// TIA Portal V18 export
FUNCTION_BLOCK "SearchArea_2doors"   // FB8, LAD
{ S7_Optimized_Access := 'TRUE' }
VERSION : 0.1
// stored: AutoNumber true, IsIECCheckEnabled false, IsRetainMemResEnabled false, MemoryReserve 100, SetENOAutomatically false, UDAEnableTagReadback false
   VAR_INPUT
      SB1 : Bool;
      SB2 : Bool;
      Door1 : Bool;
      Door2 : Bool;
      "E-Stop" : Bool;
      SearchArea_Time : Time := T#5m;
      Reset : Bool;
   END_VAR
   VAR
      SearchArea_Timer { S7_SetPoint := 'True'} : TON_TIME;
      SearchArea_Status : Int;   // 0:未搜索;1:搜索中;2:搜索完成;
      "Step" { S7_SetPoint := 'True'} : Int;
      Error { ExternalAccessible := 'False'; ExternalVisible := 'False'; ExternalWritable := 'False'} : Struct
         All { ExternalAccessible := 'False'; ExternalVisible := 'False'; ExternalWritable := 'False'} : Bool;   // 搜索总故障
         StartFail { ExternalAccessible := 'False'; ExternalVisible := 'False'; ExternalWritable := 'False'} : Bool;   // 搜索启动失败，请确认未按下搜索按钮2或未关闭门1或门2
         WrongSequence1 { ExternalAccessible := 'False'; ExternalVisible := 'False'; ExternalWritable := 'False'} : Bool;   // 搜索顺序错误，此时应按下搜索按钮2，请勿按搜索按钮1或关闭门1或门2
         WrongSequence2 { ExternalAccessible := 'False'; ExternalVisible := 'False'; ExternalWritable := 'False'} : Bool;   // 搜索顺序错误，此时应关闭门1，请勿按搜索按钮1或搜索按钮2或门2
         WrongSequence3 { ExternalAccessible := 'False'; ExternalVisible := 'False'; ExternalWritable := 'False'} : Bool;   // 搜索顺序错误，此时应关闭门2，请勿按搜索按钮1或搜索按钮2或打开门1
         Timeout { ExternalAccessible := 'False'; ExternalVisible := 'False'; ExternalWritable := 'False'} : Bool;   // 搜索超时
      END_STRUCT;
   END_VAR
   VAR_TEMP   // added for the SCL form of the ladder/FBD networks
      _w1 : Bool;
   END_VAR
BEGIN

REGION Network 1: 搜索破坏
   // 搜索完成后，当搜索按钮按下，门被打开，急停按钮按下，搜索状态设置为未搜索
   // 需与客户确认破坏条件是否包含搜索按钮和急停？
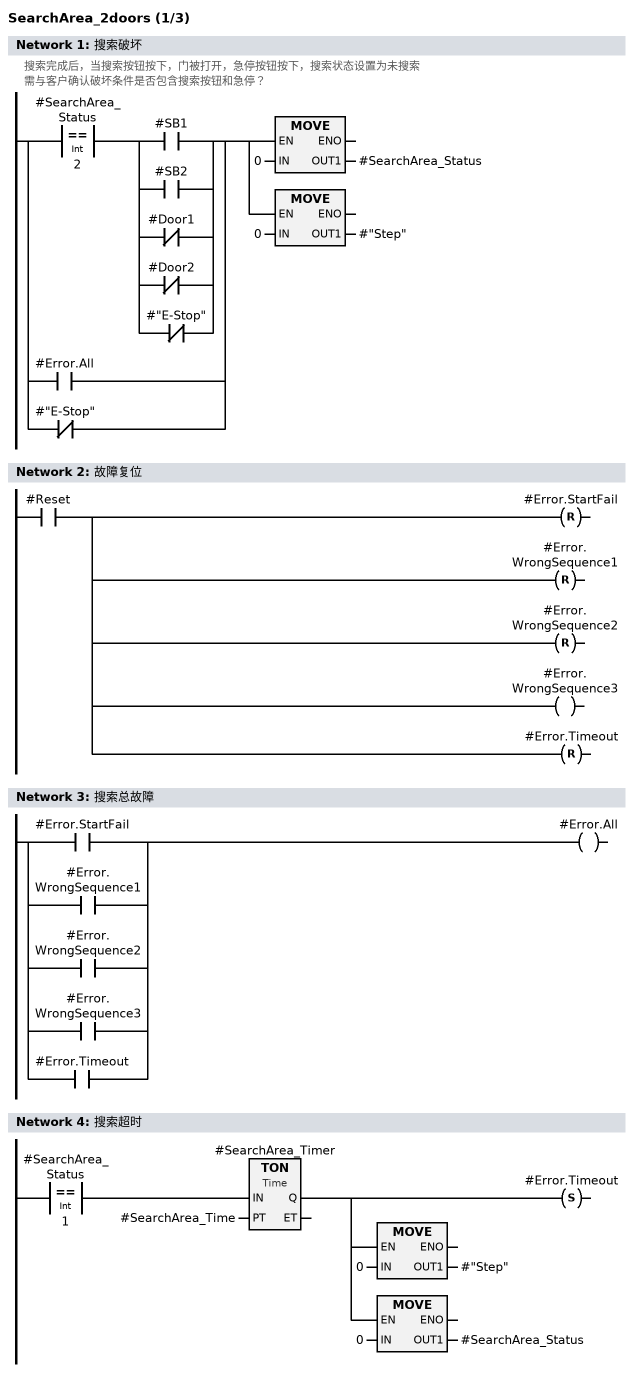
   RUNG wire#powerrail
      { S7_Templates := "SrcType := Int" } EQ_Contact(in1 := #SearchArea_Status, in2 := 2)
      wire#w1
      Contact( #SB1 )
      wire#w2
      Move(in := 0, out1 => #SearchArea_Status)
   END_RUNG
   RUNG wire#w1
      Contact( #SB2 )
   END_RUNG wire#w2
   RUNG wire#w1
      I_Contact( #Door1 )
   END_RUNG wire#w2
   RUNG wire#w1
      I_Contact( #Door2 )
   END_RUNG wire#w2
   RUNG wire#w1
      I_Contact( #"E-Stop" )
   END_RUNG wire#w2
   RUNG wire#powerrail
      Contact( #Error.All )
   END_RUNG wire#w2
   RUNG wire#powerrail
      I_Contact( #"E-Stop" )
   END_RUNG wire#w2
   RUNG wire#w2
      Move(in := 0, out1 => #"Step")
   END_RUNG
   // the same network as SCL:
   #_w1 := ((#SearchArea_Status = 2) AND (#SB1 OR #SB2 OR NOT #Door1 OR NOT #Door2 OR NOT #"E-Stop")) OR #Error.All OR NOT #"E-Stop";
   IF #_w1 THEN
       #SearchArea_Status := 0;
       #"Step" := 0;
   END_IF;
END_REGION

REGION Network 2: 故障复位
   RUNG wire#powerrail
      Contact( #Reset )
      wire#w1
      R_Coil( #Error.StartFail )
   END_RUNG
   RUNG wire#w1
      R_Coil( #Error.WrongSequence1 )
   END_RUNG
   RUNG wire#w1
      R_Coil( #Error.WrongSequence2 )
   END_RUNG
   RUNG wire#w1
      Coil( #Error.WrongSequence3 )
   END_RUNG
   RUNG wire#w1
      R_Coil( #Error.Timeout )
   END_RUNG
   // the same network as SCL:
   IF #Reset THEN
       #Error.StartFail := FALSE;
       #Error.WrongSequence1 := FALSE;
       #Error.WrongSequence2 := FALSE;
   END_IF;
   #Error.WrongSequence3 := #Reset;
   IF #Reset THEN #Error.Timeout := FALSE; END_IF;
END_REGION

REGION Network 3: 搜索总故障
   RUNG wire#powerrail
      Contact( #Error.StartFail )
      wire#w1
      Coil( #Error.All )
   END_RUNG
   RUNG wire#powerrail
      Contact( #Error.WrongSequence1 )
   END_RUNG wire#w1
   RUNG wire#powerrail
      Contact( #Error.WrongSequence2 )
   END_RUNG wire#w1
   RUNG wire#powerrail
      Contact( #Error.WrongSequence3 )
   END_RUNG wire#w1
   RUNG wire#powerrail
      Contact( #Error.Timeout )
   END_RUNG wire#w1
   // the same network as SCL:
   #Error.All := #Error.StartFail OR #Error.WrongSequence1 OR #Error.WrongSequence2 OR #Error.WrongSequence3 OR #Error.Timeout;
END_REGION

REGION Network 4: 搜索超时
   RUNG wire#powerrail
      { S7_Templates := "SrcType := Int" } EQ_Contact(in1 := #SearchArea_Status, in2 := 1)
      { S7_Templates := "time_type := Time" } #SearchArea_Timer.TON(pt := #SearchArea_Time, et =>)
      wire#w1
      S_Coil( #Error.Timeout )
   END_RUNG
   RUNG wire#w1
      Move(in := 0, out1 => #"Step")
   END_RUNG
   RUNG wire#w1
      Move(in := 0, out1 => #SearchArea_Status)
   END_RUNG
   // the same network as SCL:
   #SearchArea_Timer(IN := #SearchArea_Status = 1, PT := #SearchArea_Time);   // TON
   IF #SearchArea_Timer.Q THEN
       #Error.Timeout := TRUE;
       #"Step" := 0;
       #SearchArea_Status := 0;
   END_IF;
END_REGION

REGION Network 5: 按下SB1，开始搜索
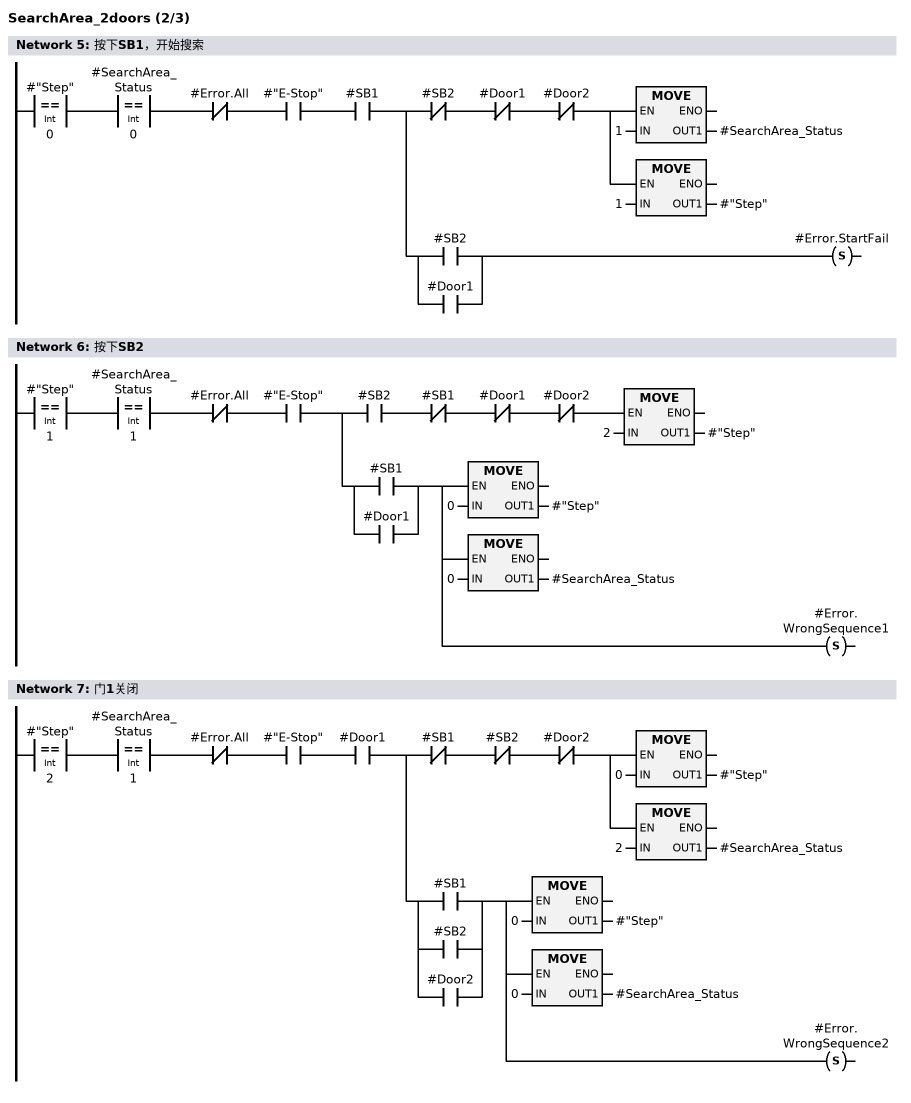
   RUNG wire#powerrail
      { S7_Templates := "SrcType := Int" } EQ_Contact(in1 := #"Step", in2 := 0)
      { S7_Templates := "SrcType := Int" } EQ_Contact(in1 := #SearchArea_Status, in2 := 0)
      I_Contact( #Error.All )
      Contact( #"E-Stop" )
      Contact( #SB1 )
      wire#w1
      I_Contact( #SB2 )
      I_Contact( #Door1 )
      I_Contact( #Door2 )
      wire#w2
      Move(in := 1, out1 => #SearchArea_Status)
   END_RUNG
   RUNG wire#w2
      Move(in := 1, out1 => #"Step")
   END_RUNG
   RUNG wire#w1
      Contact( #SB2 )
      wire#w3
      S_Coil( #Error.StartFail )
   END_RUNG
   RUNG wire#w1
      Contact( #Door1 )
   END_RUNG wire#w3
   // the same network as SCL:
   #_w1 := (#"Step" = 0) AND (#SearchArea_Status = 0) AND NOT #Error.All AND #"E-Stop" AND #SB1;
   IF #_w1 AND NOT #SB2 AND NOT #Door1 AND NOT #Door2 THEN
       #SearchArea_Status := 1;
       #"Step" := 1;
   END_IF;
   IF #_w1 AND (#SB2 OR #Door1) THEN #Error.StartFail := TRUE; END_IF;
END_REGION

REGION Network 6: 按下SB2
   RUNG wire#powerrail
      { S7_Templates := "SrcType := Int" } EQ_Contact(in1 := #"Step", in2 := 1)
      { S7_Templates := "SrcType := Int" } EQ_Contact(in1 := #SearchArea_Status, in2 := 1)
      I_Contact( #Error.All )
      Contact( #"E-Stop" )
      wire#w1
      Contact( #SB2 )
      I_Contact( #SB1 )
      I_Contact( #Door1 )
      I_Contact( #Door2 )
      Move(in := 2, out1 => #"Step")
   END_RUNG
   RUNG wire#w1
      Contact( #SB1 )
      wire#w2
      Move(in := 0, out1 => #"Step")
   END_RUNG
   RUNG wire#w1
      Contact( #Door1 )
   END_RUNG wire#w2
   RUNG wire#w2
      Move(in := 0, out1 => #SearchArea_Status)
   END_RUNG
   RUNG wire#w2
      S_Coil( #Error.WrongSequence1 )
   END_RUNG
   // the same network as SCL:
   #_w1 := (#"Step" = 1) AND (#SearchArea_Status = 1) AND NOT #Error.All AND #"E-Stop";
   IF #_w1 AND #SB2 AND NOT #SB1 AND NOT #Door1 AND NOT #Door2 THEN #"Step" := 2; END_IF;
   IF #_w1 AND (#SB1 OR #Door1) THEN
       #"Step" := 0;
       #SearchArea_Status := 0;
       #Error.WrongSequence1 := TRUE;
   END_IF;
END_REGION

REGION Network 7: 门1关闭
   RUNG wire#powerrail
      { S7_Templates := "SrcType := Int" } EQ_Contact(in1 := #"Step", in2 := 2)
      { S7_Templates := "SrcType := Int" } EQ_Contact(in1 := #SearchArea_Status, in2 := 1)
      I_Contact( #Error.All )
      Contact( #"E-Stop" )
      Contact( #Door1 )
      wire#w1
      I_Contact( #SB1 )
      I_Contact( #SB2 )
      I_Contact( #Door2 )
      wire#w2
      Move(in := 0, out1 => #"Step")
   END_RUNG
   RUNG wire#w2
      Move(in := 2, out1 => #SearchArea_Status)
   END_RUNG
   RUNG wire#w1
      Contact( #SB1 )
      wire#w3
      Move(in := 0, out1 => #"Step")
   END_RUNG
   RUNG wire#w1
      Contact( #SB2 )
   END_RUNG wire#w3
   RUNG wire#w1
      Contact( #Door2 )
   END_RUNG wire#w3
   RUNG wire#w3
      Move(in := 0, out1 => #SearchArea_Status)
   END_RUNG
   RUNG wire#w3
      S_Coil( #Error.WrongSequence2 )
   END_RUNG
   // the same network as SCL:
   #_w1 := (#"Step" = 2) AND (#SearchArea_Status = 1) AND NOT #Error.All AND #"E-Stop" AND #Door1;
   IF #_w1 AND NOT #SB1 AND NOT #SB2 AND NOT #Door2 THEN
       #"Step" := 0;
       #SearchArea_Status := 2;
   END_IF;
   IF #_w1 AND (#SB1 OR #SB2 OR #Door2) THEN
       #"Step" := 0;
       #SearchArea_Status := 0;
       #Error.WrongSequence2 := TRUE;
   END_IF;
END_REGION

REGION Network 8: 门2关闭
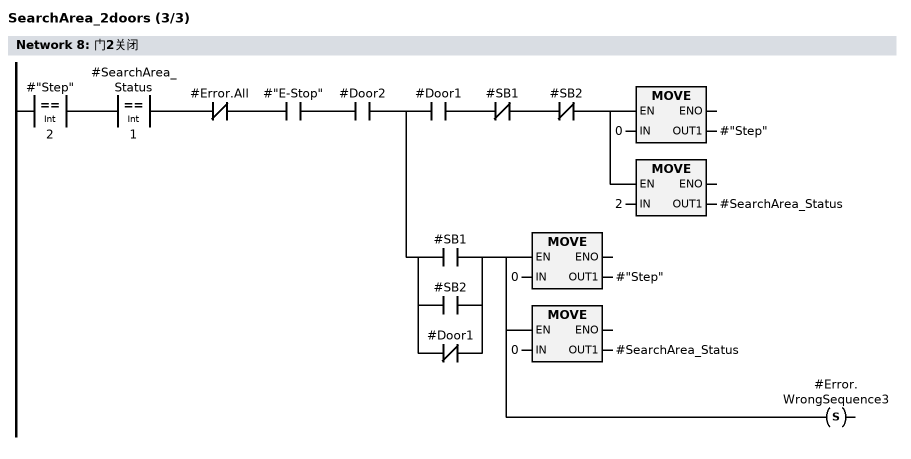
   RUNG wire#powerrail
      { S7_Templates := "SrcType := Int" } EQ_Contact(in1 := #"Step", in2 := 2)
      { S7_Templates := "SrcType := Int" } EQ_Contact(in1 := #SearchArea_Status, in2 := 1)
      I_Contact( #Error.All )
      Contact( #"E-Stop" )
      Contact( #Door2 )
      wire#w1
      Contact( #Door1 )
      I_Contact( #SB1 )
      I_Contact( #SB2 )
      wire#w2
      Move(in := 0, out1 => #"Step")
   END_RUNG
   RUNG wire#w2
      Move(in := 2, out1 => #SearchArea_Status)
   END_RUNG
   RUNG wire#w1
      Contact( #SB1 )
      wire#w3
      Move(in := 0, out1 => #"Step")
   END_RUNG
   RUNG wire#w1
      Contact( #SB2 )
   END_RUNG wire#w3
   RUNG wire#w1
      I_Contact( #Door1 )
   END_RUNG wire#w3
   RUNG wire#w3
      Move(in := 0, out1 => #SearchArea_Status)
   END_RUNG
   RUNG wire#w3
      S_Coil( #Error.WrongSequence3 )
   END_RUNG
   // the same network as SCL:
   #_w1 := (#"Step" = 2) AND (#SearchArea_Status = 1) AND NOT #Error.All AND #"E-Stop" AND #Door2;
   IF #_w1 AND #Door1 AND NOT #SB1 AND NOT #SB2 THEN
       #"Step" := 0;
       #SearchArea_Status := 2;
   END_IF;
   IF #_w1 AND (#SB1 OR #SB2 OR NOT #Door1) THEN
       #"Step" := 0;
       #SearchArea_Status := 0;
       #Error.WrongSequence3 := TRUE;
   END_IF;
END_REGION
END_FUNCTION_BLOCK
